FUNCTION_BLOCK PLOT_JSON_TIMESERIES
  {SET_ATTRIBUTE(OpcUa, SERVICE)}
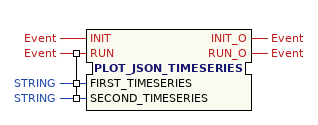
  EVENT_INPUT
    INIT;
    RUN WITH FIRST_TIMESERIES, SECOND_TIMESERIES;
  END_EVENT
  EVENT_OUTPUT
    INIT_O;
    RUN_O;
  END_EVENT
  VAR_INPUT
    FIRST_TIMESERIES : STRING; {SET_ATTRIBUTE(OpcUa, Variable.RUN)}
    SECOND_TIMESERIES : STRING; {SET_ATTRIBUTE(OpcUa, Variable.RUN)}
  END_VAR
END_FUNCTION_BLOCK
